// TIA Portal V21 export
TYPE "Std_eResponseToValveModeSet"
   STRUCT
      reserved { ExternalVisible := 'False'} : Int;
      invalid_SetValveMode { ExternalVisible := 'False'} : Int := 1;
      invalid_SetAppControl { ExternalVisible := 'False'} : Int := 2;
      invalid_SetAppOption { ExternalVisible := 'False'} : Int := 3;
      invalid_SetPointValue1 { ExternalVisible := 'False'} : Int := 4;
      invalid_SetPointValue2 { ExternalVisible := 'False'} : Int := 5;
      invalid_configuration { ExternalVisible := 'False'} : Int := 6;
      access_denied_WebConfig { ExternalVisible := 'False'} : Int := 10;
      access_denied_saving_parametrisation { ExternalVisible := 'False'} : Int := 11;
      no_license_for_this_MA { ExternalVisible := 'False'} : Int := 12;
      all_licenses_in_use { ExternalVisible := 'False'} : Int := 13;
      invalid_license_file { ExternalVisible := 'False'} : Int := 14;
      no_valve_detected { ExternalVisible := 'False'} : Int := 15;
      valve_self_calibration_running { ExternalVisible := 'False'} : Int := 16;
      no_TransferMode_with_this_FB { ExternalVisible := 'False'} : Int := 1020;
      preparing_for_start { ExternalVisible := 'False'} : Int := 1031;
      starting { ExternalVisible := 'False'} : Int := 1032;
      MA_running { ExternalVisible := 'False'} : Int := 1033;
      Transfermode_running { ExternalVisible := 'False'} : Int := 1034;
      stopping { ExternalVisible := 'False'} : Int := 1035;
      all_MAs_stopped { ExternalVisible := 'False'} : Int := 1036;
      acknowledge_needed { ExternalVisible := 'False'} : Int := 1037;
      failure { ExternalVisible := 'False'} : Int := 1038;
      preparing_for_acknowledge { ExternalVisible := 'False'} : Int := 1040;
      acknowledging { ExternalVisible := 'False'} : Int := 1041;
      all_errors_acknowledged { ExternalVisible := 'False'} : Int := 1042;
      failure_still_active { ExternalVisible := 'False'} : Int := 1043;
      no_Communication { ExternalVisible := 'False'} : Int := 1050;
      FB_not_enabled { ExternalVisible := 'False'} : Int := 1051;
   END_STRUCT;
END_TYPE
